// TIA Portal V16 export
// export: Created 2022-02-04T14:40:23.6911611Z, ExportSetting WithDefaults, DisplayName Totally Integrated Automation Portal, DisplayVersion V16 Update 1, DisplayName TIA Portal Version Control Interface, DisplayVersion V16, DisplayName TIA Portal Openness, DisplayVersion V16, DisplayName SINAMICS Startdrive Advanced, DisplayVersion V16 Update 5, DisplayName SINAMICS Startdrive G130, G150, S120, S150, SINAMICS MV, S210, DisplayVersion V16 Update 5, DisplayName SINAMICS Startdrive G110M, G120, G120C, G120D, G120P, G115D, DisplayVersion V16 Update 5, DisplayName STEP 7 Professional, DisplayVersion V16, DisplayName STEP 7 Safety, DisplayVersion V16, DisplayName WinCC Advanced, DisplayVersion V16, DisplayName SIMATIC Visualization Architect, DisplayVersion V16
VAR_GLOBAL   // PLC tag table "Стандартная таблица переменных"
   "K1-112 2L1" AT %I0.0 : Bool;   // Реле безопастности К10 ОСНОВНАЯ напряжение управления
   "K1-113/1 3L1" AT %I0.1 : Bool;   // Реле безопастности К11 концевики группа 211,212,213,214
   "K1-113/2 4L1" AT %I0.2 : Bool;   // Реле безопастности К21 группа 221,222,224,225,231-235,311,312,313-317
   "K1-113/3 5L1" AT %I0.3 : Bool;   // Релле безопасности К31 группа 321,322,324
   "k1-113/4 6L1" AT %I0.4 : Bool;   // Релле безопасности К41 группа 331,332-337
   Varalla AT %I0.5 : Bool;   // резерв
   Varalla1 AT %I0.6 : Bool;   // резерв
   Varalla2 AT %I0.7 : Bool;   // резерв
   "211K1/211K2" AT %I1.0 : Bool;   // М211 включен сигналы
   "212K1" AT %I1.1 : Bool;   // Контактор К1 Включен М212 сигналы
   "213K1" AT %I1.2 : Bool;   // контактор К1 Включен М213 сигналы
   "311K1/311K2" AT %I1.3 : Bool;   // М311 включен сигналы
   Varalla3 AT %I1.4 : Bool;   // резерв
   Varalla4 AT %I1.5 : Bool;   // резерв
   Varalla5 AT %I1.6 : Bool;   // резерв
   Varalla6 AT %I1.7 : Bool;   // резерв
   "221K1" AT %I2.0 : Bool;   // М221 включен сигналы
   "222K1" AT %I2.1 : Bool;   // Контактор К1 Включен М222 сигналы
   "223K1" AT %I2.2 : Bool;   // Обратная связь
   "224K1" AT %I2.3 : Bool;   // М224 включен сигналы
   "225K1" AT %I2.4 : Bool;   // Контактор К1 Включен М225 сигналы
   "330K1" AT %I2.5 : Bool;   // Контактор К1 Включен М330 сигнал
   Varalla8 AT %I2.6 : Bool;   // резерв
   Varalla9 AT %I2.7 : Bool;   // резерв
   "231K1" AT %I3.0 : Bool;   // Контактор К1 Включен М231 сигналы
   "232K1" AT %I3.1 : Bool;   // Контактор К1- Включен М232 сигналы
   "233K1" AT %I3.2 : Bool;   // Контактор К1- Включен М233 сигналы
   "234K1" AT %I3.3 : Bool;   // М234 включен сигналы
   "235K1/235K2" AT %I3.4 : Bool;   // М235 включен сигналы
   Varalla10 AT %I3.5 : Bool;   // резерв
   Varalla11 AT %I3.6 : Bool;   // резерв
   Varalla12 AT %I3.7 : Bool;   // резерв
   "214K1" AT %I4.0 : Bool;   // М214 включен сигналы
   "312K1" AT %I4.1 : Bool;   // М312 включен сигналы
   "313K1/313K2" AT %I4.2 : Bool;   // М313 включен сигналы
   "314K1" AT %I4.3 : Bool;   // М314 включен сигналы
   "315K1" AT %I4.4 : Bool;   // М315 включен сигналы
   "316K1" AT %I4.5 : Bool;   // М316 включен сигналы
   "317K1" AT %I4.6 : Bool;   // Контактор К1 включен М317 сигналы
   Varalla13 AT %I4.7 : Bool;   // резерв
   "321K1/321K2" AT %I5.0 : Bool;   // М321 включен сигналы
   "322K1/322K2" AT %I5.1 : Bool;   // М322 включен сигналы
   "323K1/323K2" AT %I5.2 : Bool;   // М323 включен сигнал
   "K1-324U.1" AT %I5.3 : Bool;   // ПЧТ 324 в работе сигналы
   "325K1" AT %I5.4 : Bool;   // Контактор К1 М325 сигнал
   Varalla15 AT %I5.5 : Bool;   // резерв
   Varalla16 AT %I5.6 : Bool;   // резеов
   Varalla17 AT %I5.7 : Bool;   // резерв
   "331K1" AT %I6.0 : Bool;   // М331 включен сигналы
   "332K1" AT %I6.1 : Bool;   // Контактор К1- включен М332 сигналы
   "333K1" AT %I6.2 : Bool;   // Контактор К1 -включен М333 сигналы
   "334K1" AT %I6.3 : Bool;   // Контактор К1- включен М334 сигналы
   "335K1" AT %I6.4 : Bool;   // Контактор К1- включен М335 сигналы
   "336K1" AT %I6.5 : Bool;   // Контактор К1- включен М336 сигналы
   "337K1" AT %I6.6 : Bool;   // Контактор К1-включен М337 сигнал
   "K1-323U1" AT %I6.7 : Bool;   // ПЧТ 312 в работе сигналы
   "K1-212U1" AT %I7.0 : Bool;   // ПЧТ 212 в работе сигналы
   "K1-213U1" AT %I7.1 : Bool;   // ПЧТ 213 в работе сигналы
   "K1-215U1" AT %I7.2 : Bool;   // ПЧТ 215 в работе сигналы
   "K1-222U1" AT %I7.3 : Bool;   // ПЧТ 222 в работе сигналы
   "K1-225U1" AT %I7.4 : Bool;   // Пчт 225 в работе сигналы
   "K1-231U1" AT %I7.5 : Bool;   // ПЧТ 231 в работе сигналы
   "K1-233U1" AT %I7.6 : Bool;   // ПЧТ 233 в работе сигналы
   "K1-317U1" AT %I7.7 : Bool;   // ПЧТ 317 в работе сигналы
   "K1-332U1" AT %I8.0 : Bool;   // ПЧТ 332 в работе сигналы
   "K1-333U1" AT %I8.1 : Bool;   // ПЧТ 333 в работе сигналы
   "K1-334U1" AT %I8.2 : Bool;   // ПЧТ 334 в работе сигналы
   "K1-335U1" AT %I8.3 : Bool;   // ПЧТ 335 в работе сигналы
   "K1-336U1" AT %I8.4 : Bool;   // ПЧТ 336 в работе сигналы
   "K1-223U1" AT %I8.5 : Bool;   // ПЧТ М223 в работе сигнал
   "K1-324U1" AT %I8.6 : Bool;   // ПЧТ М324 в работе сигнал
   "K1-325U1" AT %I8.7 : Bool;   // ПЧТ М325 в работе сигнал
   "K1/112-S1" AT %I9.0 : Bool;   // Состояние концевика 112S1 сигналы
   "K1/112-S2" AT %I9.1 : Bool;   // Состояние концевика 112S2 сигналы
   "K1/112-S3" AT %I9.2 : Bool;   // Состояние концевика 112S3 сигналы
   Varalla22 AT %I9.3 : Bool;   // резерв
   "K1/113-S11" AT %I9.4 : Bool;   // Состояние концевиков 113S11 сигналы
   "K1/113-S12" AT %I9.5 : Bool;   // Состояние концевиков 113S12 сигналы
   "k1/113-S13" AT %I9.6 : Bool;   // Состояние концевиков 113S13 сигналы
   "FC 323.1" AT %I9.7 : Bool;   // Датчик блокировки поштучной
   "FC 323.2" AT %I10.0 : Bool;   // Датчик на останов основной горки
   "FC 223.1" AT %I10.1 : Bool;   // Начало зоны оценки
   "FC 223.2" AT %I10.2 : Bool;   // Конец зоны оценки
   "FC 223.3" AT %I10.3 : Bool;   // Сброс доски в брак
   FC_323_1 AT %I10.4 : Bool;   // резерв
   Key_Faser AT %I10.5 : Bool;   // индуктивник положения поштучной выдачи
   Varalla30 AT %I10.6 : Bool;   // резерв
   Varalla31 AT %I10.7 : Bool;   // резерв
   "Lift Upp" AT %I11.0 : Bool;   // Лифт вниз
   "Lift Down" AT %I11.1 : Bool;   // Лифт в верх
   "sloi doski" AT %I11.2 : Bool;   // Слой доски 1
   "sloi doski2" AT %I11.3 : Bool;   // Слой доски 2
   "doska v priymke elevator" AT %I11.4 : Bool;   // Доска в приямке элеватора
   koncevik1 AT %I11.5 : Bool;   // концевик 1(середина приемного транспортера)
   koncevik2 AT %I11.6 : Bool;   // концевик 2 (вилы лифта приемного транспортера)
   "nakloniy transporter" AT %I11.7 : Bool;   // наклонный транспортер датчик
   "1,8m" AT %I12.0 : Bool;   // 1,8 длинна
   "2,1m" AT %I12.1 : Bool;   // 2,1 длинна
   "2,4m" AT %I12.2 : Bool;   // 2,4 длинна
   "2,7m" AT %I12.3 : Bool;   // 2,7 длинна
   "3,0m" AT %I12.4 : Bool;   // 3,0 длинна
   "3,3m" AT %I12.5 : Bool;   // 3,3 длинна
   "3,6m" AT %I12.6 : Bool;   // 3,6 длинна
   "3,9m" AT %I12.7 : Bool;   // 3,9 длинна
   "4,2m" AT %I13.0 : Bool;   // 4,2 длинна
   "4,5m" AT %I13.1 : Bool;   // 4,5 длинна
   "4,8m" AT %I13.2 : Bool;   // 4,8 длинна
   "5,1m" AT %I13.3 : Bool;   // 5,1 длинна
   "5,4m" AT %I13.4 : Bool;   // 5,4 длинна
   "5,7m" AT %I13.5 : Bool;   // 5,7 длинна
   "6,0m" AT %I13.6 : Bool;   // 6,0 длинна
   PodBort_1 AT %I13.7 : Bool;   // Положение подвижного борта_1
   PodBort_2 AT %I14.0 : Bool;   // Положение подвижного борта _2
   K312Fault AT %I14.1 : Bool;   // Авария частотника 312
   "S14.2" AT %I14.2 : Bool;   // Максимальная ширина доски концевик М225 зона
   "S14.3" AT %I14.3 : Bool;   // Минимальная ширина доски концевик М225 зона
   "B14.4" AT %I14.4 : Bool;   // счет доски М225 зона после бобышек
   "B14.5" AT %I14.5 : Bool;   // счет доски М225 зона после бобышек
   "K-312U1" AT %I14.6 : Bool;   // ПЧТ 312 В работе
   "S14.7" AT %I14.7 : Bool;   // заднее положение вил
   "S15.0" AT %I15.0 : Bool;   // замедление вил назад
   "S15.1" AT %I15.1 : Bool;   // замедление в перед вил
   "S15.2" AT %I15.2 : Bool;   // Переднее положение вил
   "311_S1" AT %I15.3 : Bool;   // Запрет двиджения М311
   Index AT %I15.4 : Bool;   // Индексная точка энкодера
   "B15.5" AT %I15.5 : Bool;   // вилы в верху
   "311_S2" AT %I15.6 : Bool;   // Ручное управление М311
   "B15.7" AT %I15.7 : Bool;   // вилы в низу
   FC_232_1 AT %I16.0 : Bool;   // набор слоя пакета на лифте1
   "S16.1" AT %I16.1 : Bool;   // лифт ПфМ в низу
   "S16.2" AT %I16.2 : Bool;   // лифт ПФМ в верху
   FC_225_Upor AT %I16.3 : Bool;   // датчик доски на упорах перед транспортером с бобышками
   "E16.4" AT %I16.4 : Bool;   // Уровень Гидростанции Основной
   FC_232_2 AT %I16.5 : Bool;   // Набор слоя пакета на лифте2
   KeyFazerPFM_repeater AT %I16.6 : Bool;   // Второй кейфазер на транспортер бобышек
   KeyFazerPFM AT %I16.7 : Bool;   // кейфазер для транспортера бобышек
   "B17.0" AT %I17.0 : Bool;   // наличие прокладок на М312
   "B17.1" AT %I17.1 : Bool;   // наличие прокладки в М314
   "B17.2" AT %I17.2 : Bool;   // наличие прокладки в М315
   "234.4" AT %I17.3 : Bool;   // второй датчик наличия прокладки перед каруселью
   "234.1" AT %I17.4 : Bool;   // 234.1 прокладка на выдаче(датчик)
   "234.2" AT %I17.5 : Bool;   // 234.2 прокладка максимальный слой
   "234.3" AT %I17.6 : Bool;   // 234.3 перекос прокладки (Авария)
   Fc316 AT %I17.7 : Bool;   // Датчик в конце М316 перед элеватором1
   "B18.0" AT %I18.0 : Bool;   // рейкоукладчик в верху
   "B18.1" AT %I18.1 : Bool;   // второй индуктив на позиционирование карусели
   "S18.2" AT %I18.2 : Bool;   // среднее положение рейкоукладчика
   "S18.3" AT %I18.3 : Bool;   // рейкоукладчик в низу
   "B18.4" AT %I18.4 : Bool;   // датчик положения захвата прокладки открыто
   "B18.5" AT %I18.5 : Bool;   // датчик положени захвата прокладки закрыто
   "B18.6" AT %I18.6 : Bool;   // сигнал набора слоя
   "B18.7" AT %I18.7 : Bool;   // Остановка транспортера прокладок
   "B19.0" AT %I19.0 : Bool;   // Обратный ход транспортера прокладок ДАТЧИК
   Varalla35 AT %I19.1 : Bool;   // резерв
   Varalla36 AT %I19.2 : Bool;   // резерв
   Varalla37 AT %I19.3 : Bool;   // резерв
   Varalla38 AT %I19.4 : Bool;   // резерв
   Varalla39 AT %I19.5 : Bool;   // резерв
   Varalla40 AT %I19.6 : Bool;   // резерв
   Varalla41 AT %I19.7 : Bool;   // резерв
   Varalla42 AT %I20.0 : Bool;   // резерв
   Varalla43 AT %I20.1 : Bool;   // резерв
   Varalla44 AT %I20.2 : Bool;   // резерв
   Varalla45 AT %I20.3 : Bool;   // резерв
   Varalla46 AT %I20.4 : Bool;   // резерв
   Varalla47 AT %I20.5 : Bool;   // резерв
   Varalla48 AT %I20.6 : Bool;   // резерв
   Varalla49 AT %I20.7 : Bool;   // резерв
   Varalla50 AT %I21.0 : Bool;   // резерв
   Varalla51 AT %I21.1 : Bool;   // резерв
   Varalla52 AT %I21.2 : Bool;   // резерв
   Varalla53 AT %I21.3 : Bool;   // резерв
   Varalla54 AT %I21.4 : Bool;   // резерв
   Varalla55 AT %I21.5 : Bool;   // резерв
   Varalla56 AT %I21.6 : Bool;   // резерв
   Varalla57 AT %I21.7 : Bool;   // резерв
   "B22.0" AT %I22.0 : Bool;   // доска в конце роликового транспортера(брак)
   "B22.1" AT %I22.1 : Bool;   // доска в начале роликового транспортера(брак)
   "S22.2" AT %I22.2 : Bool;   // вилы брака ПФМ в перед
   "S22.3" AT %I22.3 : Bool;   // вилы брака ПФМ назад
   "B22.4" AT %I22.4 : Bool;   // лифт брака ПФМ в верху
   "B22.5" AT %I22.5 : Bool;   // лифт брака ПФМ в низу
   "B22.6" AT %I22.6 : Bool;   // Слой на вилах брака ПФМ
   "FC 22.7" AT %I22.7 : Bool;   // Счет доски слоя на пфм Брака
   "B23.0" AT %I23.0 : Bool;   // Пакет на основном разгрузочном транспортере3
   "B23.1" AT %I23.1 : Bool;   // пакет на разгрузочном транспортере 2
   M324Sync AT %I23.2 : Bool;   // индуктив синхронизации М 324
   Varalla60 AT %I23.3 : Bool;   // резерв
   Varalla61 AT %I23.4 : Bool;   // резерв
   Varalla62 AT %I23.5 : Bool;   // резерв
   "FC 23.6" AT %I23.6 : Bool;   // Упоры подняты ПФМ брака
   "FC 23.7" AT %I23.7 : Bool;   // Упоры опущены ПФМ брака
   S76 AT %I24.0 : Bool;   // стоповая кнопка OP1
   "S76.1" AT %I24.1 : Bool;   // Включение напряжения управления
   "S76.2" AT %I24.2 : Bool;   // Подтверждение ошибки
   "S76.3" AT %I24.3 : Bool;   // Гидравлика линии в положении включено
   "E76.4" AT %I24.4 : Bool;   // Старт гидравлики
   "S76.5" AT %I24.5 : Bool;   // авто включение и выключение загрузчика ( режим авто всей загрузки)
   "S76.6" AT %I24.6 : Bool;   // авто М211 приемный транспортер
   "E76.7" AT %I24.7 : Bool;   // вперед М211 приемный транспортер в автомате
   "S77.0" AT %I25.0 : Bool;   // авто М222 горка
   "E77.1" AT %I25.1 : Bool;   // вперед М222 горка в автомате
   "S77.2" AT %I25.2 : Bool;   // Квитирование зоны 1(от горки до ПФМ)
   "S77.3" AT %I25.3 : Bool;   // Квитирование зоны выгрузки
   "S77.4" AT %I25.4 : Bool;   // Квитирование зоны 2 (ПФМ брака)
   "S77.5" AT %I25.5 : Bool;   // авто режим зоны 1( включено, выключено) ( от горки до ПФМ)
   "S77.6" AT %I25.6 : Bool;   // Выдвинуть упоры поштучника
   "E77.7" AT %I25.7 : Bool;   // Убрать упоры поштучника
   "S78.0" AT %I26.0 : Bool;   // Вилы выдвинуть
   "E78.1" AT %I26.1 : Bool;   // Вилы задвинуть
   "S78.2" AT %I26.2 : Bool;   // Вилы опустить
   "E78.3" AT %I26.3 : Bool;   // Вилы поднять
   "S78.4" AT %I26.4 : Bool;   // Лифт опустить
   "E78.5" AT %I26.5 : Bool;   // Лифт поднять
   "S78.6" AT %I26.6 : Bool;   // рейкоукладчик вниз
   "E78.7" AT %I26.7 : Bool;   // рейкоукладчик вверх
   "S79.0" AT %I27.0 : Bool;   // принудительно завершить сборку пакета
   "S79.1" AT %I27.1 : Bool;   // авто подача прокладки(включен,выключен)
   "E79.2" AT %I27.2 : Bool;   // резерв
   "S79.3" AT %I27.3 : Bool;   // авто режим ПФМ брака (включено,выключено)
   "S79.4" AT %I27.4 : Bool;   // Сброс с рольганга(брака) вперпед
   "S79.5" AT %I27.5 : Bool;   // Транспортер набора слоя ( брака) вперед
   "S79.6" AT %I27.6 : Bool;   // вилы( брака) вперед
   "E79.7" AT %I27.7 : Bool;   // вилы( брака) назад
   "S80.0" AT %I28.0 : Bool;   // Упоры слоя ПФМ( брака)
   "E80.1" AT %I28.1 : Bool;   // Упоры слоя ПФМ( брака)
   "S80.2" AT %I28.2 : Bool;   // Лифт ПФМ(брака) опустить
   "E80.3" AT %I28.3 : Bool;   // Лифт ПФМ(брака) поднять
   "S80.4" AT %I28.4 : Bool;   // поднять, опустить Подвижный борт(М235)
   "S80.5" AT %I28.5 : Bool;   // вперед подвижный борт(М235)
   "E80.6" AT %I28.6 : Bool;   // назад подвижный борт(М235)
   "S80.7" AT %I28.7 : Bool;
   Varalla106 AT %I29.0 : Bool;   // резерв
   Varalla107 AT %I29.1 : Bool;   // резерв
   Varalla108 AT %I29.2 : Bool;   // резерв
   Varalla109 AT %I29.3 : Bool;   // резерв
   Varalla110 AT %I29.4 : Bool;   // резерв
   Varalla111 AT %I29.5 : Bool;   // резерв
   Varalla112 AT %I29.6 : Bool;   // резерв
   Varalla113 AT %I29.7 : Bool;   // резерв
   "S82.0" AT %I30.0 : Bool;   // Стоп ОР2
   "S81.1" AT %I30.1 : Bool;   // Приемный транспортер вперед ОР2
   "E82.2" AT %I30.2 : Bool;   // Приемный транспортер назад ОР2
   "S82.3" AT %I30.3 : Bool;   // Авто загрузка включена,выключена ОР2
   "S82.4" AT %I30.4 : Bool;   // Лифт загрузки поднять ОР2
   "E82.5" AT %I30.5 : Bool;   // Лифт загрузки опустить ОР2
   "S82.6" AT %I30.6 : Bool;   // Наклонный транспортер авто ОР2
   "E82.7" AT %I30.7 : Bool;   // Авто наклонный транспортер вперед ОР2
   "S83.0" AT %I31.0 : Bool;   // Ленточный транспортер удаления прокладок назад ОР2
   "E83.1" AT %I31.1 : Bool;   // Ленточный транспортер удаления прокладок вперед ОР2
   "E83.2" AT %I31.2 : Bool;   // Горка прокладок 1 авто ОР2
   "E83.3" AT %I31.3 : Bool;   // Горка прокладок 1 вперед ОР2(авто)
   "S83.4" AT %I31.4 : Bool;   // Квитирование зоны 1 ОР2
   Varalla114 AT %I31.5 : Bool;   // резерв
   Varalla115 AT %I31.6 : Bool;   // резерв
   Varalla116 AT %I31.7 : Bool;   // резерв
   "S84.0" AT %I32.0 : Bool;   // Стоп ОР3
   "S84.1" AT %I32.1 : Bool;   // Транспортер М317 прокладок вперед ОР3
   "E84.2" AT %I32.2 : Bool;   // Транспортер М317 прокладок назад ОР3
   "S84.3" AT %I32.3 : Bool;   // Дозированиe включено ОР3
   "S84.4" AT %I32.4 : Bool;   // авто подача прокладок включена, выключена ОР3
   "S84.5" AT %I32.5 : Bool;   // Рейкоукладчик вниз ОР3
   "E84.6" AT %I32.6 : Bool;   // Рейкоукладчик вверх ОР3
   "S84.7" AT %I32.7 : Bool;   // Открыть стакан прокладки ОР3
   "E85.0" AT %I33.0 : Bool;   // Закрыть стакан прокладки ОР3
   "S85.1" AT %I33.1 : Bool;
   "E85.2" AT %I33.2 : Bool;
   "S85.3" AT %I33.3 : Bool;   // авто горка прокладок 2,3 ОР3
   "E85.4" AT %I33.4 : Bool;   // горка 2,3 прокладок вперед(авто) ОР3
   "S85.5" AT %I33.5 : Bool;   // М234 назад ОР3
   "E85.6" AT %I33.6 : Bool;   // М234 вперед транспортер прокладок перед крючками ОР3
   "S85.7" AT %I33.7 : Bool;   // Квитирование зоны прокладок ОР3
   "S86.0" AT %I34.0 : Bool;   // Лифт ПФМ вниз ОР3
   "E86.1" AT %I34.1 : Bool;   // ЛИфт ПФМ вверх ОР3
   "S86.2" AT %I34.2 : Bool;   // Ролики лифта ПФМ вперед ОР3
   "S86.3" AT %I34.3 : Bool;   // ПФМ Основное Авто включено, выключено ОР3
   "S86.4" AT %I34.4 : Bool;   // Подтверждение неисправности ОР3
   "S86.5" AT %I34.5 : Bool;   // датчик
   Varalla117 AT %I34.6 : Bool;   // резерв
   Varalla118 AT %I34.7 : Bool;   // резерв
   "S87.0" AT %I35.0 : Bool;   // Кнопка брака ОР1.1
   "S87.1" AT %I35.1 : Bool;   // Горка авто ОР1.1
   "E87.2" AT %I35.2 : Bool;   // Горка ОР1.1 (авто)
   "S87.3" AT %I35.3 : Bool;   // датчик перекоса перед плавниками
   "S87.4" AT %I35.4 : Bool;   // набор ковра перед плавниками
   Varalla119 AT %I35.5 : Bool;   // резерв
   Varalla120 AT %I35.6 : Bool;   // резерв
   Varalla121 AT %I35.7 : Bool;   // резерв
   "S88.0" AT %I36.0 : Bool;   // Стоп ОР4
   "K3.3" AT %I36.1 : Bool;   // работа подвижного борта ОР4
   "S88.2" AT %I36.2 : Bool;   // Выкатной транспортер 1 ПФМ назад ОР4
   "E88.3" AT %I36.3 : Bool;   // Выкатной транспортер 1 ПФМ вперед ОР4
   "S88.4" AT %I36.4 : Bool;   // Выкатной транспортер 2 ПФМ назад ОР4
   "S88.5" AT %I36.5 : Bool;   // Выкатной транспортер 2 ПФМ вперед ОР4
   "E88.6" AT %I36.6 : Bool;   // резерв ОР4
   "S88.7" AT %I36.7 : Bool;   // резерв ОР4
   "S89.0" AT %I37.0 : Bool;   // Выкатной транспортер 3 ПФМ назад ОР4
   "S89.1" AT %I37.1 : Bool;   // Выкатной транспортер 3 ПФМ вперед ОР4
   "S89.2" AT %I37.2 : Bool;   // Квитирование ОР4
   "S89.3" AT %I37.3 : Bool;   // датчик ОР4
   Varalla122 AT %I37.4 : Bool;   // резерв ОР4
   Varalla123 AT %I37.5 : Bool;   // резерв ОР4
   Varalla124 AT %I37.6 : Bool;   // резерв ОР4
   Varalla125 AT %I37.7 : Bool;   // резерв ОР4
   "S90.0" AT %I38.0 : Bool;   // Стоп ОР5
   "S90.1" AT %I38.1 : Bool;   // М331 вперед ленточный транспортер брака ОР5
   "S90.2" AT %I38.2 : Bool;   // М332 вперед сбрасыватель рольганга брака ОР5
   Varalla126 AT %I38.3 : Bool;   // резерв
   "S90.4" AT %I38.4 : Bool;   // Вилы ПФМ брака назад ОР5
   "E90.5" AT %I38.5 : Bool;   // Вилы ПФМ брака вперед ОР5
   "S90.6" AT %I38.6 : Bool;   // Опустить упоры формирования слоя на ПФМ брака ОР5
   "E90.7" AT %I38.7 : Bool;   // Поднять упоры формирования слоя на ПФМ брака ОР5
   "S91.0" AT %I39.0 : Bool;   // Лифт брака ПФМ опустить ОР5
   "E91.1" AT %I39.1 : Bool;   // Лифт брака ПФМ поднять ОР5
   "S91.2" AT %I39.2 : Bool;   // квитирование ПФМ 2
   Varalla127 AT %I39.3 : Bool;   // резерв
   Varalla128 AT %I39.4 : Bool;   // резерв
   Varalla129 AT %I39.5 : Bool;   // резерв
   Varalla130 AT %I39.6 : Bool;   // резерв
   Varalla131 AT %I39.7 : Bool;   // резерв
   "K1-212U" AT %QW512 : Int;
   "K1-213U" AT %QW514 : Int;
   "K1-215U" AT %QW516 : Int;
   "K1-222U" AT %QW518 : Int;
   "K1-225U" AT %QW520 : Int;
   "K1-231U" AT %QW522 : Int;
   "K1-233U" AT %QW524 : Int;
   "K1-317U" AT %QW526 : Int;
   "K1-332U" AT %QW528 : Int;
   "K1-333U" AT %QW530 : Int;
   "K1-334U" AT %QW532 : Int;
   "K1-335U" AT %QW534 : Int;
   "K1-336U" AT %QW536 : Int;
   "K1-223U" AT %QW538 : Int;
   "k1-323U" AT %QW540 : Int;
   "K1-325U" AT %QW542 : Int;
   "K1-112x1" AT %Q0.0 : Bool;   // релле Сирены
   "Sk1-113" AT %Q0.1 : Bool;   // разрешение на запуск релле К10 безопастность
   "K1-113X1" AT %Q0.2 : Bool;   // разрешение на запуск релле К11 безопастность
   "K1-113X2" AT %Q0.3 : Bool;   // разрешение на запуск релле К21 безопастность
   "K1-113X3" AT %Q0.4 : Bool;   // разрешение на запуск релле К31 безопастность
   "K1-113X4" AT %Q0.5 : Bool;   // разрешение на запуск релле К41 безопастность
   Varalla65 AT %Q0.6 : Bool;   // резерв
   Varalla66 AT %Q0.7 : Bool;   // резерв
   "K1-211X1" AT %Q1.0 : Bool;   // М211 вперед загрузочный транспортер
   "K1-211X1.1" AT %Q1.1 : Bool;   // М211 назад загрузочный транспортер
   "K1-212X1" AT %Q1.2 : Bool;   // контактор К1-212 ПЧТ запуск лифт
   "K1-212X1.1" AT %Q1.3 : Bool;   // Растормаживание М212 лифт
   "K1-213X1" AT %Q1.4 : Bool;   // контактор К1-213 ПЧТ запуск наклонный транспортер
   "K1-311X1" AT %Q1.5 : Bool;   // запуск ленточного транспортера удалителя прокладок M311
   Varalla68 AT %Q1.6 : Bool;   // резерв
   Varralla69 AT %Q1.7 : Bool;   // резерв
   "K1-221X1" AT %Q2.0 : Bool;   // запуск М221 гидростанция1
   "K1-222X1" AT %Q2.1 : Bool;   // Запуск контактора К1-222 ПЧТ основной элеватор
   "K1-223X1" AT %Q2.2 : Bool;   // запуск М223 Цепной после поштучника
   "K1-224X1" AT %Q2.3 : Bool;   // запуск М224 выдвинуть упоры поштучника
   "K1-224-x1.1" AT %Q2.4 : Bool;   // запуск М224 задвинуть упоры поштучника
   "K1-225X1" AT %Q2.5 : Bool;   // включение контактора К1-225 ПЧТ транспортер бобышек
   "K1-231X1" AT %Q2.6 : Bool;   // включение контактора К1-231 ПЧТ ролики торцовочные
   "K1-232X1" AT %Q2.7 : Bool;   // включение контактора К1-232 ПЧТ Лифт ПФМ
   "K1-232X1.1" AT %Q3.0 : Bool;   // Тормоз Лифта ПФМ
   "K1-233X1" AT %Q3.1 : Bool;   // включение контактора К1-233 ПЧТ вилы ПФМ
   "K1-234X1" AT %Q3.2 : Bool;   // запуск М234 транспортер прокладок перед крючками ПФМ
   "K1-235X1" AT %Q3.3 : Bool;   // запуск М235 вперед подвижный борт
   "K1-214X1" AT %Q3.4 : Bool;   // запуск М214 транспортер загрузки прокладок
   "K1-330X1" AT %Q3.5 : Bool;   // запуск М330 контактора лента брака2
   "K1-312X1" AT %Q3.6 : Bool;   // запуск М312 первая горка прокладок
   "K1-313X1" AT %Q3.7 : Bool;   // запуск М313 вперед транспортер прокладок после первой горки
   "K1-313X1.1" AT %Q4.0 : Bool;   // запуск М313 назад транспортера прокладок после первой горки
   "K1-314X1" AT %Q4.1 : Bool;   // запуск М314 горка прокладок 2
   "K1-315X1" AT %Q4.2 : Bool;   // запуск М315 горка прокладок 3
   "K1-316X1" AT %Q4.3 : Bool;   // запуск М316 транспортер загрузки прокладок в горку 2
   "K1-317X1" AT %Q4.4 : Bool;   // включение контактора К1-317 ПЧТ основной транспортер прокладок
   "K1-317X1.1" AT %Q4.5 : Bool;   // тормоз М317
   "K1-321X1" AT %Q4.6 : Bool;   // запуск М321 вперед выкатной транспортер ПФМ
   "K1-321X1.1" AT %Q4.7 : Bool;   // запуск М321 назад выкатной транспортер ПФМ
   "K1-322X1" AT %Q5.0 : Bool;   // запуск М322 вперед выкатной транспортер ПФМ2
   "K1-322X1.1" AT %Q5.1 : Bool;   // Запуск М322 назад выкатной транспортер ПФМ2
   "K1-323X1" AT %Q5.2 : Bool;   // Запуск контактора М323 маленький после элеватора
   "K1-325U2" AT %Q5.3 : Bool;   // Старт ПЧТ М325 набор слоя основной
   "K1-324U2" AT %Q5.4 : Bool;   // команда на ПЧТ вперед М324 выгрузка покета выкатной ПФМ3
   "K1-324U2.2" AT %Q5.5 : Bool;   // команда на ПЧТ назад М324 выгрузка покета выкатной ПФМ3
   "K1-325X1" AT %Q5.6 : Bool;   // Включение контактора К1-325 ПЧТ набор слоя основной
   "K1-235X1.1" AT %Q5.7 : Bool;   // запуск М235 назад подвижный борт
   "K1-331X1" AT %Q6.0 : Bool;   // запуск М331 ленточный транспортер брака
   "K1-332x1" AT %Q6.1 : Bool;   // включение контактора К1-332 ПЧТ сбрасыватель с рольганга (брак)
   "K1--333X1" AT %Q6.2 : Bool;   // включение контактора К1-333 ПЧТ рольганг (брака)
   "K1-334X1" AT %Q6.3 : Bool;   // включение контактора К1-334 ПЧТ транспортер сбора слоя ПФМ брака
   "K1-335X1" AT %Q6.4 : Bool;   // включение контактора К1-335 ПЧТ вилы ПФМ брака
   "K1-336X1" AT %Q6.5 : Bool;   // Включение контактора К1-336 ПЧТ лифт ПФМ брака
   "K1-336X1.1" AT %Q6.6 : Bool;   // Тормоз М336 лифта ПФМ брака
   "K1-337K1" AT %Q6.7 : Bool;   // Контактор пуска Гирдростанции ПФМ Брака
   Varalla70 AT %Q7.0 : Bool;   // резерв
   "K1-312U2" AT %Q7.1 : Bool;   // Старт ПЧТ 312
   Varalla72 AT %Q7.2 : Bool;   // резерв
   Varalla73 AT %Q7.3 : Bool;   // резерв
   Varalla74 AT %Q7.4 : Bool;   // резерв
   Varalla75 AT %Q7.5 : Bool;   // резерв
   Varalla76 AT %Q7.6 : Bool;   // резерв
   Varalla77 AT %Q7.7 : Bool;   // резерв
   "K1-212U2" AT %Q8.0 : Bool;   // старт ПЧТ М212
   "K1-212U2.2" AT %Q8.1 : Bool;   // Реверс ПЧТ М212
   "K1-213U2" AT %Q8.2 : Bool;   // Старт ПЧТ М213
   "K1-215U2" AT %Q8.3 : Bool;   // Старт ПЧТ 232
   "K1-215U2.2" AT %Q8.4 : Bool;   // Реверс ПЧТ 232
   "K1-222U2" AT %Q8.5 : Bool;   // Старт ПЧТ 222
   "K1-225U2" AT %Q8.6 : Bool;   // Старт ПЧТ 225
   "K1-231U2" AT %Q8.7 : Bool;   // Старт ПЧТ 231
   "K1-233U2" AT %Q9.0 : Bool;   // Старт ПЧТ 233
   "K1-233U2.2" AT %Q9.1 : Bool;   // Реверс ПЧТ 233
   "K1-223U2" AT %Q9.2 : Bool;   // Старт ПЧТ 223
   "K1-332U2" AT %Q9.3 : Bool;   // Старт ПЧТ 332
   "K1-333U2" AT %Q9.4 : Bool;   // Старт ПЧТ 333
   "K1-334U2" AT %Q9.5 : Bool;   // Старт ПЧТ 334
   "K1-335U2" AT %Q9.6 : Bool;   // Старт ПЧТ 335
   "K1-335U2.2" AT %Q9.7 : Bool;   // Реверс ПЧТ 335
   "K1-336U2" AT %Q10.0 : Bool;   // Стасрт ПЧТ 336
   "K1-336U2.2" AT %Q10.1 : Bool;   // Реверс ПЧТ 336
   "K1-317U2" AT %Q10.2 : Bool;   // Старт ПЧТ 317
   "K1-317U2.2" AT %Q10.3 : Bool;   // Реверс ПЧТ 317
   Y223_1 AT %Q12.0 : Bool;   // переворот доски вверх
   Y223_2 AT %Q12.1 : Bool;   // переворот доски вниз
   Y223_3 AT %Q12.2 : Bool;   // сброс в брак вниз
   Y223_4 AT %Q12.3 : Bool;   // сброс в брак вверх
   Y323_1 AT %Q12.4 : Bool;   // упоры перед поштучкой вверх
   Y323_2 AT %Q12.5 : Bool;   // упоры перед поштучкой вниз
   Upor_brak_up AT %Q12.6 : Bool;   // упоры ПФМ брака вверх
   Upor_brak_down AT %Q12.7 : Bool;   // упоры ПФМ брака вниз
   "Y223.3" AT %Q13.0 : Bool;   // перепускной клапан маленькая гидростанция
   "Y223.4" AT %Q13.1 : Bool;   // перепускной клапан маленькая гидростанция
   Varalla89 AT %Q11.6 : Bool;   // резерв
   Varalla90 AT %Q11.7 : Bool;   // резерв
   "K1-323U2" AT %Q10.4 : Bool;   // Старт ПЧТ 323
   "Y12.1" AT %Q10.5 : Bool;   // резерв
   Varalla91 AT %Q10.6 : Bool;   // резерв
   Varalla92 AT %Q10.7 : Bool;   // резерв
   Varalla93 AT %Q11.0 : Bool;   // резерв
   Varalla94 AT %Q11.1 : Bool;   // резерв
   Varalla95 AT %Q11.2 : Bool;   // резерв
   Varalla96 AT %Q11.3 : Bool;   // резерв
   "Y13.0" AT %Q11.4 : Bool;
   "Y13.1" AT %Q11.5 : Bool;
   "Y13.2" AT %Q13.2 : Bool;
   "Y13.3" AT %Q13.3 : Bool;
   "Y13.4" AT %Q13.4 : Bool;
   "Y13.5" AT %Q13.5 : Bool;
   "Y13.6" AT %Q13.6 : Bool;
   "Y13.7" AT %Q13.7 : Bool;
   Line1_1 AT %Q14.0 : Bool;   // вилы вниз
   Line1_2 AT %Q14.1 : Bool;   // вилы вверх
   Line2_1 AT %Q14.2 : Bool;   // упоры перед поштучкой вверх
   Line2_2 AT %Q14.3 : Bool;   // упоры перед поштучкой вниз
   Line3_1 AT %Q14.4 : Bool;   // подвижный борт опустить
   Line3_2 AT %Q14.5 : Bool;   // подвижный борт поднять
   Line4_1 AT %Q14.6 : Bool;   // выдача прокладки вниз
   Line4_2 AT %Q14.7 : Bool;   // выдача прокладки вверх
   Perepusk AT %Q15.0 : Bool;   // перепускной клапан большая гидростанция
   Line5_1 AT %Q15.1 : Bool;   // каретка прокладки вниз
   Line5_2 AT %Q15.2 : Bool;   // каретка прокладки вверх
   Line6_1 AT %Q15.3 : Bool;   // ложементы закрыть
   Line6_2 AT %Q15.4 : Bool;   // ложементы открыть
   Varalla100 AT %Q15.5 : Bool;   // резерв
   Varalla101 AT %Q15.6 : Bool;   // резерв
   Varalla102 AT %Q15.7 : Bool;   // резерв
   "H76.0" AT %Q16.0 : Bool;   // Напряжение управления включено (лампочка) ОР1
   "H76.1" AT %Q16.1 : Bool;   // потверждение аварии (лампочка) ОР1
   "H76.2" AT %Q16.2 : Bool;   // Гидравлика линии в положении включено (лампочка) ОР1
   "H76.3" AT %Q16.3 : Bool;   // авто включение и выключение загрузчика ( режим авто всей загрузки) (лампочка)ОР1
   "H76.4" AT %Q16.4 : Bool;   // разгрусчик открыт (лапмочка) ОР1
   "H76.5" AT %Q16.5 : Bool;   // Квитирование ПФМ 1 (лапмочка)ОР1
   "H76.6" AT %Q16.6 : Bool;   // Квитирование (лампочка)ОР1
   "H76.7" AT %Q16.7 : Bool;   // Квитирование ПФМ 2 (лампочка)ОР1
   "H77.0" AT %Q17.0 : Bool;   // ПФМ 1 авто включено ( лампочка)ОР1
   "H77.1" AT %Q17.1 : Bool;   // авто подача прокладки(включен,выключен) (лампочка)ОР1
   "H77.2" AT %Q17.2 : Bool;   // Авто ПФМ 2 включен (лампочка)ОР1
   Varalla132 AT %Q17.3 : Bool;   // резерв ОР1
   Varalla133 AT %Q17.4 : Bool;   // резерв ОР1
   Varalla134 AT %Q17.5 : Bool;   // резерв ОР1
   Varalla135 AT %Q17.6 : Bool;   // резерв ОР1
   Varalla136 AT %Q17.7 : Bool;   // резерв ОР1
   "H78.0" AT %Q18.0 : Bool;   // Авто загрузка включена,выключена ОР2 (лампочка)
   "H78.1" AT %Q18.1 : Bool;   // квитирование загрузки (лампочка)ОР2
   Varalla137 AT %Q18.2 : Bool;   // резерв
   Varalla138 AT %Q18.3 : Bool;   // резерв
   "A78.4" AT %Q18.4 : Bool;   // Авто подачи прокладок включен (лампочка)ОР3
   "A78.5" AT %Q18.5 : Bool;   // Квитирование прокладок (лампочка)ОР3
   "A78.6" AT %Q18.6 : Bool;   // Авто ПФМ 1 включен ( лампочка) ОР3
   "H78.7" AT %Q18.7 : Bool;   // Авария (лампочка)ОР3
   "H79.0" AT %Q19.0 : Bool;   // Квитирование выгрузки (лампочка) ОР4
   Pakkauspuristin AT %Q19.1 : Bool;
   "A79.2" AT %Q19.2 : Bool;   // резерв
   "A79.3" AT %Q19.3 : Bool;   // резерв
   "H79.4" AT %Q19.4 : Bool;   // Квитирование ПФМ2 (лампочка)
   Varalla139 AT %Q19.5 : Bool;   // резерв
   Varalla140 AT %Q19.6 : Bool;   // резерв
   Varalla141 AT %Q19.7 : Bool;   // резерв
   Lift AT %M20.0 : Bool;
   FALSE AT %M20.1 : Bool;
   M212StartDelay AT %T1 : Timer;   // Задержка перд стартом загрузки пакета на лифт
   Tag_2 AT %T2 : Timer;
   M212DownDelay AT %T3 : Timer;   // Задержка на опускания лифта вниз
   DropDelay AT %T4 : Timer;   // задержка на срабатывания датчиков сброся слоя
   m212waitAfterDrop AT %T6 : Timer;   // Задержка на сброс доски после сброса
   m213DropDelay AT %T7 : Timer;
   M212waitEmptyHole AT %T8 : Timer;   // Ожидание освобождения приямка горки загрузки
   Tag_9 AT %T9 : Timer;
   M211startDelay AT %T10 : Timer;   // задержка старта транспортера при установке пакета погрузчиком
   Tag_11 AT %T11 : Timer;
   Tag_12 AT %T12 : Timer;
   Tag_13 AT %T13 : Timer;
   Tag_14 AT %T14 : Timer;
   Tag_15 AT %T15 : Timer;
   Tag_16 AT %T16 : Timer;
   Tag_17 AT %T17 : Timer;
   Tag_18 AT %T18 : Timer;
   Tag_5 AT %M0.0 : Bool;
   Tag_61 AT %M0.1 : Bool;
   Tag_62 AT %T19 : Timer;
   NaprUpr AT %M0.6 : Bool;   // меркер напряжения управления
   Tag_19 AT %C1 : Counter;
   Tag_20 AT %C2 : Counter;
   HodVil2 AT %M1.2 : Bool;
   Tag_71 AT %T5 : Timer;
   Tag_72 AT %T20 : Timer;
   Tag_73 AT %C3 : Counter;
   Fouls AT %M4.0 : Bool;
   TRUE AT %M4.1 : Bool;
   "Tag_19(1)" AT %T21 : Timer;
   M213AlarmFilter AT %T22 : Timer;
   M214AlarmFilter AT %T23 : Timer;
   "221StartDelay" AT %T24 : Timer;
   "222AlarmFilter" AT %T25 : Timer;
   "223AlarmFilter" AT %T26 : Timer;
   "332AlarmFilter" AT %T27 : Timer;
   "333AlarmFilter" AT %T28 : Timer;
   "334AlarmFilter" AT %T29 : Timer;
   "336DownDelay" AT %T30 : Timer;
   "336AlarmFilter" AT %T31 : Timer;
   "321AlarmFilter" AT %T32 : Timer;
   "322AlarmFilter" AT %T33 : Timer;
   "324AlarmFilter" AT %T34 : Timer;
   "214AlarmFiltr" AT %T35 : Timer;
   "312AlarmFiltr" AT %T36 : Timer;
   "313AlarmFilter" AT %T37 : Timer;
   "316AlarmFiltr" AT %T38 : Timer;
   "314AlarmFilter" AT %T39 : Timer;
   "234AlarmFilter" AT %T40 : Timer;
   Tag_3 AT %M4.7 : Bool;
   "224AlarmFilter" AT %T41 : Timer;
   "225AlarmFilter" AT %T42 : Timer;
   "231AlarmFilter" AT %T43 : Timer;
   "235AlarmFilter" AT %T44 : Timer;
   "311AlarmFilter" AT %T45 : Timer;
   "335AlarmFilter" AT %T46 : Timer;
   "331AlarmFilter" AT %T47 : Timer;
   "233AlarmFilter" AT %T48 : Timer;
   "337AlarmFilter" AT %T49 : Timer;
   "232AlarmFilter" AT %T50 : Timer;
   alarm AT %M2.0 : Bool;
   M323_HoldRun AT %T51 : Timer;
   Tag_1 AT %C4 : Counter;
   Tag_4 AT %T52 : Timer;
   Tag_6 AT %M2.1 : Bool;
   M323_RunTask AT %T53 : Timer;
   Tag_7 AT %T54 : Timer;
   Tag_8 AT %T55 : Timer;
   ElevatorPFM_Defective_cmd_lowering AT %M4.5 : Bool;
   Tag_21 AT %T56 : Timer;
   Tag_22 AT %M40.0 : Bool;
   Tag_23 AT %M40.1 : Bool;
   Tag_24 AT %M40.2 : Bool;
   Tag_25 AT %M40.3 : Bool;
   Tag_26 AT %M40.4 : Bool;
   Tag_27 AT %M40.5 : Bool;
   Tag_28 AT %M40.6 : Bool;
   Tag_29 AT %M40.7 : Bool;
   Tag_30 AT %M41.0 : Bool;
   Tag_31 AT %M41.1 : Bool;
   Tag_32 AT %IW544 : Word;
   Tag_33 AT %IW545 : Word;
   Tag_34 AT %M5.0 : Bool;
   Tag_35 AT %T79 : Timer;
   Tag_36 AT %T78 : Timer;
   Tag_37 AT %T80 : Timer;
   Tag_38 AT %T67 : Timer;
   Tag_39 AT %T68 : Timer;
   Tag_40 AT %T81 : Timer;
   Tag_41 AT %M5.2 : Bool;
   Tag_42 AT %T82 : Timer;
   Tag_43 AT %M5.6 : Bool;
   Tag_44 AT %T83 : Timer;
   Tag_45 AT %M5.7 : Bool;
   Tag_46 AT %T84 : Timer;
   Hill_endTask AT %T85 : Timer;
   Tag_48 AT %M6.0 : Bool;
   Tag_49 AT %M6.1 : Bool;
   Tag_50 AT %M6.2 : Bool;
   Tag_51 AT %T86 : Timer;
   Tag_52 AT %M6.3 : Bool;
   Tag_53 AT %T87 : Timer;
   Tag_54 AT %M41.2 : Bool;
   Tag_55 AT %T88 : Timer;
   Tag_56 AT %T89 : Timer;
   Tag_57 AT %M7.4 : Bool;
   Tag_58 AT %T90 : Timer;
   Tag_59 AT %T92 : Timer;
   Tag_60 AT %M7.2 : Bool;
   Tag_63 AT %T91 : Timer;
   Tag_64 AT %M4.2 : Bool;
   Tag_65 AT %M4.3 : Bool;
   Tag_66 AT %M4.4 : Bool;
   Tag_67 AT %M4.6 : Bool;
   Feed_cmd AT %M5.1 : Bool;
   Tag_69 AT %T93 : Timer;
   Tag_70 AT %M5.3 : Bool;
   Tag_74 AT %T94 : Timer;
   Tag_75 AT %M5.4 : Bool;
   Tag_76 AT %T95 : Timer;
   Tag_77 AT %IW19 : Word;
   Tag_78 AT %IB19 : Byte;
   Tag_79 AT %T96 : Timer;
   EvevatorPFM_Defective_cmd_UP AT %M41.3 : Bool;
   Tag_81 AT %T97 : Timer;
   Tag_82 AT %T98 : Timer;
   Tag_83 AT %T99 : Timer;
   Tag_84 AT %M41.4 : Bool;
   Tag_85 AT %M41.5 : Bool;
   Tag_86 AT %C5 : Counter;
   Tag_87 AT %C6 : Counter;
   StartMakeGasketLayer AT %M41.6 : Bool;
   ElevatorPFM_Defective_cmd_pushPack AT %M41.7 : Bool;
   LayerGetRidOff_flag AT %M42.0 : Bool;
   UporDispenser_permission AT %M42.1 : Bool;
   Tag_92 AT %M42.2 : Bool;
   Tag_93 AT %M42.3 : Bool;
   Tag_94 AT %T100 : Timer;
   Tag_95 AT %T101 : Timer;
   Tag_96 AT %T102 : Timer;
   Tag_97 AT %T103 : Timer;
   Tag_98 AT %T104 : Timer;
   Tag_99 AT %T105 : Timer;
   LampOp3On_Hz AT %M42.4 : Bool;
   Tag_101 AT %T106 : Timer;
   Tag_102 AT %T107 : Timer;
   LampOp3On_NoHz AT %M42.5 : Bool;
   Tag_104 AT %T108 : Timer;
   Tag_105 AT %T109 : Timer;
   Tag_106 AT %T110 : Timer;
   Tag_107 AT %T120 : Timer;
   Tag_108 AT %M10.0 : Bool;
   Tag_109 AT %T121 : Timer;
   Tag_110 AT %M10.1 : Bool;
   Tag_111 AT %T122 : Timer;
   Tag_112 AT %M10.2 : Bool;
   Tag_113 AT %T124 : Timer;
   Tag_114 AT %T111 : Timer;
   SensLineAlarms AT %M42.6 : Bool;
   CarouselManAlarms AT %M10.5 : Bool;
   UporDispenser_down AT %M42.7 : Bool;
   AlarmInfoOnly AT %M43.0 : Bool;
   FC_323_1_delayed AT %T130 : Timer;
   SensorLineRawData AT %IW12 : Word;
   "2Hz" AT %M43.1 : Bool;
   Tag_123 AT %T112 : Timer;
   Tag_124 AT %M43.2 : Bool;
   Tag_125 AT %T113 : Timer;
   Tag_126 AT %T114 : Timer;
   DelayDovodPFM AT %T115 : Timer;
   DelayStartM225 AT %T116 : Timer;
   DelayUporBrak_OFF AT %T117 : Timer;
   FC_323_1_holded AT %T118 : Timer;
   M_334_permission AT %T119 : Timer;
   BoardKickDefect_task AT %T123 : Timer;
   RunM330_M331 AT %T125 : Timer;
   RunM333 AT %T126 : Timer;
END_VAR
